// TIA Portal V19 export
TYPE "LEXCHANGETRAY_typeRoller_recieve_interface"
// stored: Access Published
   STRUCT
      logistics : "LEXCHANGETRAY_typeRoller_toLogisticsRecieve";
      workStationRoller : "LEXCHANGETRAY_typeRoller_toWorkstationRecieve";
   END_STRUCT;
END_TYPE
